TEXTLIST TL_Device
  0 = 'Choose'
  1 = 'Tested Terminal'
  2 = 'Reference Terminal'
   = ''
END_TEXTLIST

(* stored: Version 1.1.0.1, ProductVersion 3.1.4020.3
   TextList TL_Device: Id {86d357fa-e507-450e-9338-2e8573d7348a} *)
